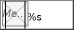
VISUALIZATION VISU_VANNE_2P_V_ACT2  // 74x30
VAR_IN_OUT
	m_Input_VANNE : BLOCK_ACTUATOR2;
END_VAR
    Rectangle (0,0 74x30), invisible if: TRUE
    Polygon (50,0)
    Polygon (50,0), colour toggle: (m_Input_VANNE.STATE_ON), invisible if: NOT (m_Input_VANNE.STATE_OFF OR m_Input_VANNE.STATE_ON) AND NOT PRG_USER.ACTU_USER.MAINTENANCE
    Rectangle (24,7 50x20), "%s", text variable: m_Input_VANNE.MNEMO
    Image (2,1 26x25), invisible if: NOT m_Input_VANNE.STATE_Nok, image: MesImages.warning
    Rectangle (5,0 20x30), invisible if: NOT (m_Input_VANNE.Autor_ON_IHM OR m_Input_VANNE.Autor_OFF_IHM) OR NOT PRG_User.ACTU_USER.MAINTENANCE
        tap m_Input_VANNE.M_ON
END_VISUALIZATION

(* stored: Version 1.1.0.1, ProductVersion 3.1.4024.10
   Visu VISU_VANNE_2P_V_ACT2: Id {ea11f137-c708-48b3-93f7-93f01ff845b6} *)
